// TIA Portal project "Software Day4 (Counters)" (V15)

(* hardware
DEVICE "S7-1200 station_1"  S7-1200 Station
   slot 0: "Rack_0"  S7-1200 Rack  Rack  V1.0
   slot 1: "PLC_1"  CPU 1215C AC/DC/Rly  6ES7 215-1BG40-0XB0  V4.2
DEVICE "HMI_1"  KTP600 Basic color PN
   slot 0: "HMI_1"  KTP600 Basic color PN  6AV6 647-0AD11-3AX0  12.0.0.0
   slot 1: "HMI_RT_1"  KTP600 Basic color PN  6AV6 647-0AD11-3AX0  12.0.0.0
   slot 5: "HMI_1.IE_CP_1"  PROFINET Interface  12.0.0.0
      slot 1: "PROFINET Interface_1"  PROFINET Interface
         slot 1: "Port_1"  Port
*)

// ===== PLC "PLC_1"  CPU 1215C AC/DC/Rly =====

VAR_GLOBAL   // PLC tag table "VAR"
   "Enter" AT %M0.1 : Bool;
   "Reset" AT %M0.3 : Bool;
   "Red Light" AT %Q0.0 : Bool;
   "Green Light" AT %Q0.1 : Bool;
   "Yellow Light" AT %Q0.2 : Bool;
   "Current  Value" AT %MW4 : Int;
   "Exit" AT %M0.2 : Bool;
   "GLO" AT %Q0.3 : Bool;
END_VAR

DATA_BLOCK "Data_block_1"   // DB3
{ S7_Optimized_Access := 'FALSE' }
VERSION : 0.1
   VAR
      Start : Bool;
      Reset : Bool;
      Current_Value : DInt;
      Red_LED : Bool;
      Stop : Bool;
      Green_LED : Bool;
      Yellow_LED : Bool;
      Fill_Valve : Bool;
      Drain_Valve : Bool;
      "Agitator Motor" : Bool;
      "Green Light" : Bool;
      "Start Batch" : Bool;
      "Stop Batch" : Bool;
      "C Value" : DInt;
      "C Out" : Bool;
      "Red Light" : Bool;
      "T  Value" : DInt;
      CV : Int;
   END_VAR
BEGIN
END_DATA_BLOCK

// folder: System blocks/Program resources

DATA_BLOCK "Cars Parking System Counter"   // DB2
{ S7_Optimized_Access := 'TRUE' }
AUTHOR : Simatic
FAMILY : IEC
NAME : CNTR
VERSION : 1.0
// stored: InstanceOfName IEC_COUNTER
"IEC_COUNTER"
BEGIN
END_DATA_BLOCK

// folder: (top level)

ORGANIZATION_BLOCK "Main"   // OB1, LAD, ProgramCycle
TITLE = "Main Program Sweep (Cycle)"
{ S7_Optimized_Access := 'TRUE' }
VERSION : 0.1
// Make a program logic for car parking system using counters.
// If no car is in parking the Green light is ON.
// If some cars are in parking the Yellow light will be ON.
// If parking is full (10 cars in stand) the Red light is ON.
   VAR_INPUT
      Initial_Call : Bool;   // Initial call of this OB
      Remanence : Bool;   // =True, if remanent data are available
   END_VAR
BEGIN

REGION Network 1
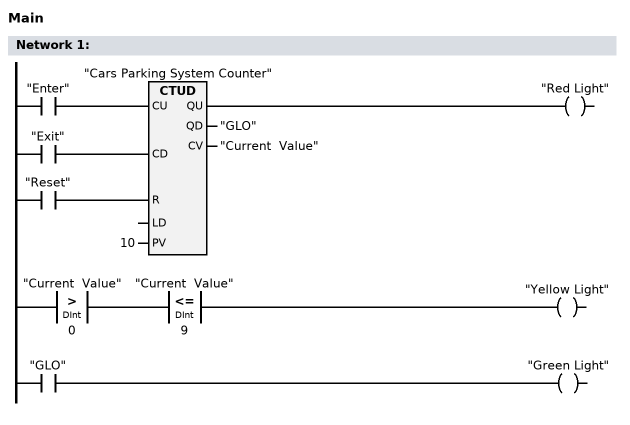
   "Cars Parking System Counter".CTUD(CU := "Enter",
                           CD := "Exit",
                           R := "Reset",
                           PV := 10,
                           QD => "GLO",
                           CV => "Current  Value");
   "Red Light" := "Cars Parking System Counter".QU;
   "Yellow Light" := ("Current  Value" > 0) AND ("Current  Value" <= 9);
   "Green Light" := "GLO";
END_REGION
END_ORGANIZATION_BLOCK

(* ===== HMI "HMI_RT_1" =====
system functions are stored by id; their names below are inferred from use
connection "HMI_Connection_1": ETHERNET, SMART_S7_1200_OMS

HMI tags "Default tag table"
   "Tag_ScreenNumber" : UInt, internal
   "Start" : Bool = PLC Enter AT %M0.1, 1 s
   "Reset" : Bool = PLC Reset AT %M0.3, 1 s
   "Current_Value" : DInt = PLC Current_Value AT %MD4, 1 s
   "Red_LED" : Bool = PLC "Red Light" AT %Q0.0, 1 s
   "Stop" : Bool = PLC Exit AT %M0.2, 1 s
   "Green_LED" : Bool = PLC "Green Light" AT %Q0.1, 1 s
   "Yellow_LED" : Bool = PLC "Yellow Light" AT %Q0.2, 1 s
   "Fill_Valve" : Bool = PLC Fill_Valve AT %Q0.6, 1 s
   "Drain_Valve" : Bool = PLC Drain_Valve AT %Q0.7, 1 s
   "Agitator Motor" : Bool = PLC "Agitator Motor" AT %Q1.0, 1 s
   "Green Light" : Bool = PLC "Green Light" AT %Q0.1, 1 s
   "Start Batch" : Bool = PLC "Start Batch" AT %M0.4, 1 s
   "Stop Batch" : Bool = PLC "Stop Batch" AT %M0.5, 1 s
   "C Value" : DInt = PLC "C Value" AT %MD5, 1 s
   "C Out" : Bool = PLC "C Out" AT %Q1.2, 1 s
   "Red Light" : Bool = PLC "Red Light" AT %Q0.0, 1 s
   "T  Value" : DInt = PLC "T  Value" AT %MD6, 1 s
   "CV" : Int = PLC CV AT %MW24, 1 s

Template "Template_1" 320x240
   Button "Exit" at 266,202 size 52x37; TextOff 'Exit'; PictureOff "ExitRuntime_KTP600_Basic_color_PN"; PictureOn "ExitRuntime_KTP600_Basic_color_PN"
      on Release: StopRuntime(0)
   Button "Alarms" at 54,202 size 52x37; TextOff 'Alarms'; PictureOff "AlarmDisplay_KTP600_Basic_color_PN"; PictureOn "AlarmDisplay_KTP600_Basic_color_PN"
      on Release: function_ef3f5d25("Alarm window_Unacknowledged", -1)
   Button "Start screen" at 1,202 size 52x37; TextOff 'Start screen'; PictureOff "NavigateHome_KTP600_Basic_color_PN"; PictureOn "NavigateHome_KTP600_Basic_color_PN"
      on Release: ActivateScreen("Root screen", 0)
   SymbolicIOField "Symbolic_IO_Field_Screen" at 69,7 size 164x24; TextOff '0'; TextOn '1'; TextList "TextList_ScreenNames"
      ProcessValue <- "Tag_ScreenNumber"
      on Change: ActivateScreenByNumber("Tag_ScreenNumber", 0)
   DateTimeField "HmiScreenItemData" at 235,19 size 85x19
   DateTimeField "HmiScreenItemData_1" at 235,0 size 85x19
   GraphicView "Logo" at 0,0 size 67x38; Picture "Logo of HMI_1"

screen "Root screen" 320x240, template "Template_1"
   on GenerateScreen: SetTag("Tag_ScreenNumber", 1)
   TextField "HmiScreenItemData" at 19,43 size 280x101; Text 'Welcome to Car Parking System'
   Button "Button_1" at 119,133 size 72x26; TextOff 'Enter'
      on Press: ActivateScreen("Screen_1", 0)

screen "Screen_1" 320x240
   Circle "Circle_1" at 240,32 size 48x48
      Appearance <- "Red_LED"
   Circle "Circle_2" at 239,107 size 48x48
      Appearance <- "Yellow_LED"
   Circle "Circle_3" at 239,170 size 48x48
      Appearance <- "Green_LED"
   Button "Button_2" at 46,144 size 50x27; TextOff 'EXIT'
      on Press: function_b14e0dd5("Stop", 0)
   Button "Button_1" at 46,80 size 50x27; TextOff 'ENTER'
      on Press: function_b14e0dd5("Start", 0)
   Button "Button_3" at 131,188 size 60x29; TextOff 'RESET'
      on Press: function_b14e0dd5("Reset", 0)
   IOField "I/O field_1" at 142,32 size 35x41; FormatPattern 99
      ProcessValue <- "CV"
*)